SUBAPPLICATION SystemTickSender (* Subapplication Type *)
  (* Standard: 61499-2 *)
  (* Version 1.0, 2026-08-07, franz *)
  PACKAGE MyLib::sys;
  IMPORT isobus::UT::Q::const::IDs::ID_NULL;
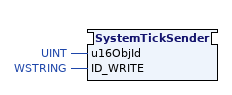
  VAR_INPUT
    u16ObjId : UINT := ID_NULL; (* Object ID *)
    ID_WRITE : WSTRING; (* OPC UA publish ID *)
  END_VAR
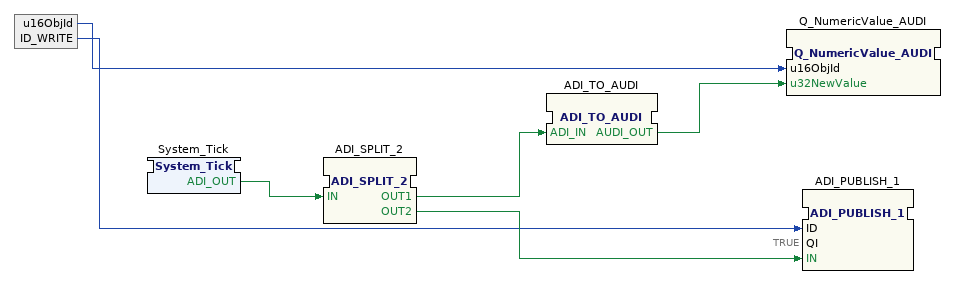
  FBS
    Q_NumericValue_AUDI : isobus::UT::Q::Q_NumericValue_AUDI;
    ADI_SPLIT_2 : adapter::events::unidirectional::ADI_SPLIT_2;
    ADI_TO_AUDI : adapter::conversion::unidirectional::ADI_TO_AUDI;
    ADI_PUBLISH_1 : adapter::net::ADI_PUBLISH_1(QI := TRUE);
  END_FBS
  SUBAPPS
    System_Tick : MyLib::sys::System_Tick;
  END_SUBAPPS
  DATA_CONNECTIONS
    u16ObjId TO Q_NumericValue_AUDI.u16ObjId;
    ID_WRITE TO ADI_PUBLISH_1.ID;
  END_CONNECTIONS
  ADAPTER_CONNECTIONS
    System_Tick.ADI_OUT TO ADI_SPLIT_2.IN;
    ADI_TO_AUDI.AUDI_OUT TO Q_NumericValue_AUDI.u32NewValue;
    ADI_SPLIT_2.OUT1 TO ADI_TO_AUDI.ADI_IN;
    ADI_SPLIT_2.OUT2 TO ADI_PUBLISH_1.IN;
  END_CONNECTIONS
END_SUBAPPLICATION
